Universal Robots PolyScope program: hookA_manager.urp

Program hookA_manager (installation=admin directory=/programs/THU_530PM createdIn=3.15.8.106339 lastSavedIn=3.15.8.106339 robotSerialNumber=2015350926)
Calibrated DH parameters: a=[0, -0.425, -0.39225, 0, 0, 0]; d=[0.089159, 0, 0, 0.10915, 0.09465, 0.0823]; alpha=[1.570796, 0, 0, 1.570796, -1.570796, 0]; deltaTheta=[0, 0, 0, 0, 0, 0]
Robot Program (runOnlyOnce=true)
  above_HookA := p[-0.27970, -0.32422, 0.12715, 2.226, -2.216, 0.000]
  offset_x := hook_index * 0.047
  above_pose_A := pose_add(above_HookA, p[0.0, -offset_x, 0.0, 0.0, 0.0, 0.0])
  at_pose_A := pose_add(above_pose_A, p[0.0, 0.0, -0.086, 0.0, 0.0, 0.0])
  Script: movel (get_inverse_kin(above_pose_A))
  Script: movel (get_inverse_kin(at_pose_A))
  Set DigitalOutput pin=digital_out[0]; digitalValue=1
  Wait Sleep waitTime=1
  Script: movel (get_inverse_kin(above_pose_A), a = 0.5, v = 0.1)
  Script: movej (get_inverse_kin(above_HookA))
  hook_index := hook_index + 1
  If hook_index ≥ num_hooks
    hook_index := 0
    Popup Message (haltProgram=false message=All Hook_A's were used! Reload Fixture inputType=Text)
